FUNCTION_BLOCK _BOOL_TestSuit EXTENDS TcUnit.FB_TestSuite
VAR
END_VAR

Placeholder();

METHOD PUBLIC Placeholder
VAR
END_VAR
TEST('Placeholder');

AssertTrue(Condition := TRUE, Message := '');

TEST_FINISHED();
END_METHOD

END_FUNCTION_BLOCK

(* stored: Version 1.1.0.1, ProductVersion 3.1.4024.12
   POU _BOOL_TestSuit: Id {04424176-653a-49ad-adf2-0c9b2705b8ed}, SpecialFunc None
   Method Placeholder: Id {ea3d6e63-a114-47ac-8ed8-933bb714da06} *)
